TYPE ST_GasSensor :
STRUCT
    nId             : INT;              // sensor ID
    eZone           : E_ZoneId;         // which zone
    rValuePPM       : REAL;             // reading in PPM
    rValueLEL       : REAL;             // reading as % LEL
    eStatus         : E_SensorStatus;   // current status
    bAlarm          : BOOL;             // alarm active
    bFault          : BOOL;             // sensor fault
    bBypassed       : BOOL;             // manually bypassed
    tLastUpdate     : TIME;             // last reading time
    sLocation       : STRING;           // physical location
END_STRUCT
END_TYPE

(* stored: Version 1.1.0.1, ProductVersion 3.1.4024.16
   DUT ST_GasSensor: Id {fb214846-bbe6-43e2-b518-c5af13df3fe0} *)
